VAR_GLOBAL CONSTANT
	None	: Result := 0; // No result or end of iteration.
	Ok		: Result := 1; // Generic success.
	Error	: Result := -1; // Generic error.
END_VAR

(* stored: Version 1.1.0.1
   GVL GenericResult: Id {b2eaa6d1-5578-4857-afc0-b7eb6736f054} *)
